(* CODESYS project EX.project

Project tree, tasks and I/O mapping:
  Device : CODESYS Control Win V3, 3S - Smart Software Solutions GmbH, order no. 305021, version 3.5.11.30
    application Application
      libraries: Standard, * (System)
      task MainTask (cyclic, interval t#20ms, priority 1) calls PLC_PRG
      program PLC_PRG [LD]
*)

// Device/Application/PLC_PRG
PROGRAM PLC_PRG
VAR
	START : BOOL;   // INICIA TODO O PROCESSO
    STOP : BOOL;    // PARA TUDO
    SE2 : BOOL;     // SENSOR DE CAIXAS
    SE1 : BOOL;     // SENSOR DE MAÇAS
    EST1 : BOOL;    // ESTEIRA DAS MAÇAS
    EST2 : BOOL;    // ESTEIRA DAS CAIXAS
	P1: BOOL;
	P2: BOOL;
	CTU_1: CTU;
	CV1: WORD;
	P3: BOOL;
	AUX: BOOL;
	P4: BOOL;
	AUX1: BOOL;
	AUX2: BOOL;
END_VAR

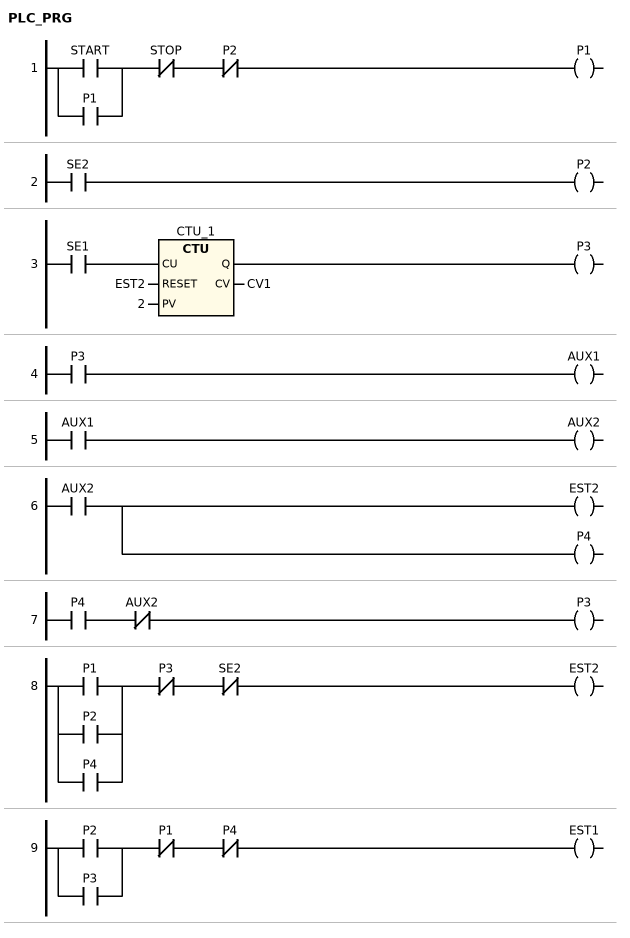
// NETWORK 1
P1 := (START OR P1) AND NOT STOP AND NOT P2;

// NETWORK 2
P2 := SE2;

// NETWORK 3
CTU_1(CU := SE1, RESET := EST2, PV := 2, CV => CV1); // CTU
P3 := CTU_1.Q;

// NETWORK 4
AUX1 := P3;

// NETWORK 5
AUX2 := AUX1;

// NETWORK 6
EST2 := AUX2;
P4 := AUX2;

// NETWORK 7
P3 := P4 AND NOT AUX2;

// NETWORK 8
EST2 := (P1 OR P2 OR P4) AND NOT P3 AND NOT SE2;

// NETWORK 9
EST1 := (P2 OR P3) AND NOT P1 AND NOT P4;

END_PROGRAM
